// TIA Portal V20 export
// export: Created 2026-07-10T11:12:34.1374805Z, ExportSetting WithDefaults, DisplayName Totally Integrated Automation Portal, DisplayVersion V20, DisplayName TIA Portal Openness, DisplayVersion V20, DisplayName TIA Portal Version Control Interface, DisplayVersion V20, DisplayName STEP 7 Professional, DisplayVersion V20, DisplayName STEP 7 Safety, DisplayVersion V20, DisplayName WinCC Basic/Comfort/Advanced, DisplayVersion V20, DisplayName WinCC Unified, DisplayVersion V20
FUNCTION_BLOCK "TankDetector"   // FB23, SCL
{ S7_Optimized_Access := 'TRUE' }
VERSION : 0.1
// stored: AutoNumber true, IsIECCheckEnabled false, IsRetainMemResEnabled false, MemoryReserve 100, SetENOAutomatically false, UDAEnableTagReadback false
   VAR_INPUT
      WeightValue : Real;
      WeightDelay : Time := T#30s;
      WeightError : Bool;
      DeadZone : Real := 0.1;
   END_VAR
   VAR_OUTPUT
      IsWeightMeasured : Bool;
      IsFeedLoaded : Bool;
      IsFeedConsumed : Bool;
      MeasuredWeight : Real;
   END_VAR
   VAR_IN_OUT
      Ref_ConsumedFeed : Real;
      Ref_LoadedFeed : Real;
      Ref_PreviousWeight : Real;
   END_VAR
   VAR
      PreviousWeight1 : Real;
      PreviousWeight2 : Real;
      TON1 { S7_SetPoint := 'True'} : TON_TIME;
      TON2 { S7_SetPoint := 'True'} : TON_TIME;
   END_VAR
BEGIN
   IF #WeightError THEN
       #IsWeightMeasured := FALSE;
       #MeasuredWeight := 0;
       RESET_TIMER(#TON1);
       RESET_TIMER(#TON2);
       RETURN;
   END_IF;

   #IsWeightMeasured := FALSE;
   #IsFeedLoaded := FALSE;
   #IsFeedConsumed := FALSE;

   IF ABS(#WeightValue - #Ref_PreviousWeight) > #DeadZone THEN
       IF #WeightValue > #Ref_PreviousWeight THEN
           #TON2(IN := TRUE,
                 PT := #WeightDelay);
           IF #TON2.Q THEN
               #IsWeightMeasured := TRUE;
               #IsFeedLoaded := TRUE;
               #MeasuredWeight := #WeightValue - #Ref_PreviousWeight;
               #Ref_LoadedFeed := #Ref_LoadedFeed + (#WeightValue - #Ref_PreviousWeight);
               #Ref_PreviousWeight := #WeightValue;
               RESET_TIMER(#TON2);
           END_IF;

           IF ABS(#WeightValue - #PreviousWeight2) > #DeadZone THEN
               RESET_TIMER(#TON2);
               #PreviousWeight2 := #WeightValue;
           END_IF;

           RESET_TIMER(#TON1);
           #PreviousWeight1 := 0;

       ELSIF #WeightValue < #Ref_PreviousWeight THEN
           #TON1(IN := TRUE,
                 PT := #WeightDelay);
           IF #TON1.Q THEN
               #IsWeightMeasured := TRUE;
               #IsFeedConsumed := TRUE;
               #MeasuredWeight := #WeightValue - #Ref_PreviousWeight;
               #Ref_ConsumedFeed := #Ref_ConsumedFeed + (#Ref_PreviousWeight - #WeightValue);
               #Ref_PreviousWeight := #WeightValue;
               RESET_TIMER(#TON1);
           END_IF;

           IF ABS(#WeightValue - #PreviousWeight1) > #DeadZone THEN
               RESET_TIMER(#TON1);
               #PreviousWeight1 := #WeightValue;
           END_IF;

           RESET_TIMER(#TON2);
           #PreviousWeight2 := 0;
       END_IF;

   ELSE
       RESET_TIMER(#TON1);
       RESET_TIMER(#TON2);
       #PreviousWeight1 := 0;
       #PreviousWeight2 := 0;
   END_IF;
END_FUNCTION_BLOCK
